// TIA Portal project "DPIS_main_project" (V17)

(* hardware
DEVICE "S7-1200 station_1"  S7-1200 Station
   slot 0: "Rack_0"  S7-1200 Rack  Rack  V1.0
   slot 1: "PLC_1"  CPU 1212C DC/DC/DC  6ES7 212-1AE40-0XB0  V4.5
   slot 2: "AI 8x13BIT_1"  6ES7 231-4HF32-0XB0  V2.1
   slot 101: "CM 1242-5"  CM 1242-5  6GK7 242-5DX30-0XE0  V1.0
*)

// ===== PLC "PLC_1"  CPU 1212C DC/DC/DC =====

VAR_GLOBAL   // PLC tag table "Default tag table"
   "mValveRightUSensor" AT %M0.0 : Bool;
   "mValveLeftUSensor" AT %M0.1 : Bool;
   "mValveLaserSensor1" AT %M0.2 : Bool;
   "mValveLaserSensor2" AT %M0.3 : Bool;
   "mValveLaserSensor3" AT %M0.4 : Bool;
   "qValveRightUSensor" AT %Q0.0 : Bool;
   "qValveLeftUSensor" AT %Q0.1 : Bool;
   "qValveLaserSensor1" AT %Q0.2 : Bool;
   "qValveLaserSensor2" AT %Q0.3 : Bool;
   "qValveLaserSensor3" AT %Q0.4 : Bool;
   "iRightUSensor" AT %I0.0 : Bool;
   "iLeftUSensor" AT %I0.1 : Bool;
   "mRightUSensor" AT %M0.5 : Bool;
   "mLeftUSensor" AT %M0.6 : Bool;
   "iLaserSensor1" AT %IW68 : Word;
   "iLaserSensor2" AT %IW70 : Word;
   "iLaserSensor3" AT %IW72 : Word;
   "iTempSensor1" AT %IW74 : Word;
   "iTempSensor2" AT %IW76 : Word;
   "iTempSensor3" AT %IW78 : Word;
   "mLaserSensor1" AT %MW2 : Word;
   "mLaserSensor2" AT %MW4 : Word;
   "mLaserSensor3" AT %MW6 : Word;
   "mTempSensor1" AT %MW8 : Word;
   "mTempSensor2" AT %MW10 : Word;
   "mTempSensor3" AT %MW12 : Word;
   "dpTempWB11" AT %IW132 : Word;
   "dpTempWB12" AT %IW134 : Word;
   "dpPalletcarSpeed" AT %IW136 : Word;
END_VAR

ORGANIZATION_BLOCK "Main"   // OB1, LAD, ProgramCycle
TITLE = "Main Program Sweep (Cycle)"
{ S7_Optimized_Access := 'TRUE' }
VERSION : 0.1
   VAR_INPUT
      Initial_Call : Bool;   // Initial call of this OB
      Remanence : Bool;   // =True, if remanent data are available
   END_VAR
BEGIN

REGION Network 2 (SCL)
   //Memory M0.0 value assign to Q0.0  ::  Right ultrasound sensor
   "qValveRightUSensor" := "mValveRightUSensor";
   //Memory M0.1 value assign to Q0.1  ::  Left ultrasound sensor
   "qValveLeftUSensor" := "mValveLeftUSensor";
   //Memory M0.2 value assign to Q0.2  ::  First laser sensor
   "qValveLaserSensor1" := "mValveLaserSensor1";
   //Memory M0.3 value assign to Q0.3  ::  Second laser sensor
   "qValveLaserSensor2" := "mValveLaserSensor2";
   //Memory M0.4 value assign to Q0.4  ::  Third laser sensor
   "qValveLaserSensor3" := "mValveLaserSensor3";
END_REGION
END_ORGANIZATION_BLOCK